DATA_BLOCK "DBHandControllerMC1"
{ S7_Optimized_Access := 'TRUE' }
VERSION : 0.1
NON_RETAIN
"FB_BasicHandController"

BEGIN

END_DATA_BLOCK

